FUNCTION_BLOCK ZONE_MDL (* HVAC Zone Model *)
  (* Standard: 61499-1; Classification: Simulation; ApplicationDomain: HVAC; Function: Zone Model *)
  (* Version 0.0, 2006-04-10, JHC, Holobloc Inc *)
  (* Compiler header: package fb.rt.hvac; *)
  (* Compiler Java Sun JDK 1.5.0 *)
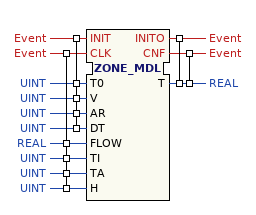
  EVENT_INPUT
    INIT WITH T0, V, AR, DT; (* Initialization Request *)
    CLK WITH FLOW, TI, H, TA; (* Simulation Clock *)
  END_EVENT
  EVENT_OUTPUT
    INITO WITH T; (* INIT completed *)
    CNF WITH T; (* Simulation step completed *)
  END_EVENT
  VAR_INPUT
    T0 : UINT := 70; (* Initial Temperature, deg F *)
    V : UINT := 5000; (* Zone volume, cu ft *)
    AR : UINT := 20; (* Wall A/R, BTU/hr/deg F *)
    DT : UINT; (* CLK cycle time, sec *)
    FLOW : REAL; (* Air Flow, CFM *)
    TI : UINT; (* Inlet Temperature, deg F *)
    TA : UINT; (* Outside Temperature, deg F *)
    H : UINT; (* Heat Load, BTU/hr *)
  END_VAR
  VAR_OUTPUT
    T : REAL; (* Zone Temperature, deg F *)
  END_VAR
  VAR
    VCV : REAL; (* Multiplier for heat load and net wall heat gain *)
    FV : REAL; (* Multiplier for (F/V) term *)
  END_VAR
  ALGORITHM INIT IN ST: (* Initialization algorithm *)
T := T0;
VCV := DT/3600.0/V/0.018;
FV := DT/60.0/V;
INITO.serviceEvent(this);
  END_ALGORITHM
  ALGORITHM CLK IN ST: (* Simulation Step algorithm *)
T := T + FV*FLOW*(TI-T) + VCV*(H+AR*(TA-T));
CNF.serviceEvent(this);
  END_ALGORITHM
END_FUNCTION_BLOCK
